FUNCTION TryConvert_LWORD_TO_BOOL : BOOL
VAR_INPUT
	in : LWORD;
	out : REFERENCE TO BOOL;
END_VAR

out := LWORD_TO_BOOL(in);
TryConvert_LWORD_TO_BOOL := TRUE;

END_FUNCTION

(* stored: Version 1.1.0.1, ProductVersion 3.1.4024.12
   POU TryConvert_LWORD_TO_BOOL: Id {9b73019f-e00b-4ea5-93d5-9383b437a8d2}, SpecialFunc None *)
